{attribute 'reflection'} 
FUNCTION_BLOCK FB_WorkerDefGrid_Python EXTENDS FB_WorkerDefGrid IMPLEMENTS I_DeformationHandler
VAR_INPUT
END_VAR
VAR_OUTPUT
END_VAR
VAR
  // interface to py script
  fbPythonInterface : FB_PythonInterface;
  // references
  _iParamMediator : I_ParamMediator;
  
  // local copy of setttings
  _bNewJob : BOOL;  // new job was activated
  _CamGridSettings : ST_CameraGridSettings;
  _DefGridSettings : ST_DefGridSettings;
  
  // local copy of job setting
  _aJobName         : T_MaxString;
  _aJobGuid         : T_MaxString;
  _fImageWidthM     : LREAL;          // image width in [m]
  _fImageDepthM     : LREAL;          // image depth in [m]
  

  // messages
  fbMsg_PythonNotRunning : FB_MESSAGE;
END_VAR

VAR CONSTANT
  fC_DEFAULT_WOKER_POSITION : LREAL := 0.01;      // default worker position in [m]
END_VAR

METHOD PROTECTED  Attach : BOOL
VAR_INPUT
  iCT              : I_CT;                         (*container at triggered event position*)
END_VAR
VAR
  pCt : POINTER TO FB_ContainerDefGrid;
END_VAR
Attach := FALSE;
IF SUPER^.Attach(iCT:=iCT) THEN
  // OK, attached (enabled, was ok to be attached)
  IF getCtInst(iCT:=iCT, pCT=>pCt) = 0 THEN    // get specific container
    RETURN;
  END_IF
  
  // setup check
  IF _iParamMediator = 0 THEN Release(iCT:=iCT); LogError('Invalid param mediator'); RETURN; END_IF
  
  // Additional worker checks
  // - do we have a valid job? used mode?
  IF _CamGridSettings.eCameraMode > E_CameraMode.NoCorrection AND (iCT.pJob = 0 OR NOT _bJobActive) THEN
    pCt^.AbortDeformation(sReason:='No valid job', Src:=_pEcSrc^);
     Release(iCT:=iCT);
     
  ELSIF _CamGridSettings.eCameraMode > E_CameraMode.NoCorrection THEN
    // OK attach
    // -- only create ct if a deformation is active
    IF CreateDefCt(iCT:=iCT) THEN
        // set state
        pCt^.StartScript(iDeformationHandler:=THIS^);
        // attached
        Attach := TRUE;
    END_IF
  ELSE
    ; // ignore attach
  END_IF
ELSE
  // parent attach failed
END_IF
END_METHOD

(*
  Create/Release virtual ct in deformation handlers.
  :return: TRUE if success
*)
METHOD PRIVATE CreateDefCt : BOOL;
VAR_INPUT
  iCT : I_CT;
END_VAR
IF iCT = 0 THEN RETURN; END_IF

IF _CamGridSettings.eCameraMode >= E_CameraMode.Live THEN
  IF fbPythonInterface.RegisterCT(iCT.pCT^.nMemIndex) THEN
    CreateDefCt := TRUE;
  ELSE
    _pAttachedCt^.AbortDeformation(sReason:='Could not register to script', Src:=_pEcSrc^);
  END_IF
ELSE
  CreateDefCt := TRUE;
END_IF
END_METHOD

METHOD DeleteCachedCt : BOOL
VAR_INPUT
	iCT	: I_CT;
END_VAR
DeleteDefCt(iCT:=iCT);
END_METHOD

(*
  Delete/Release virtual ct in deformation handlers.
  :return: TRUE if sucess
*)
METHOD DeleteDefCt : BOOL
VAR_INPUT
  iCT : I_CT;
END_VAR
IF iCT = 0 THEN RETURN; END_IF

IF _CamGridSettings.eCameraMode >= E_CameraMode.Live THEN
  IF fbPythonInterface.RemoveCT(iCT.pCT^.nMemIndex) THEN
    DeleteDefCt := TRUE;
  ELSE
    LogError('Could not delete ct in script');
  END_IF
END_IF
END_METHOD

METHOD Init
VAR_INPUT
  iWorkerParams : I_WorkerParams;
  pMsgConfig : POINTER TO ST_MSG_CONFIG;         // message config
  fPrintResolution : LREAL := 1;                 // print(head) resolution in [dpi]
  fSubPxResolution : LREAL := 1;                 // SubPixel resolution [SubPx], resolution factor (fI_PrintResolution*fI_SubPxResolution=>Output resolution)
  bParallelCT : BOOL;                            // Support parallel processing of CTs
END_VAR
SUPER^.Init(iWorkerParams:=iWorkerParams, pMsgConfig:=pMsgConfig, fPrintResolution:=fPrintResolution, fSubPxResolution:=fSubPxResolution, bParallelCT:=bParallelCT);

// Init messages
fbMsg_PythonNotRunning.pI_MsgConfig := _pMsgConfigExt;
fbMsg_PythonNotRunning.iI_MsgLocation := ePr_BLK_PU;
fbMsg_PythonNotRunning.iI_MsgNumber := eC_DMAX_DEF_SCRIPT_NOT_RUNNING;
END_METHOD

METHOD InitWorkerPython
VAR_INPUT
  aScriptPath : T_MaxString;                     // path to cmd scripts
  //aAmsLocalHost : T_AmsNetID;                    // Ams netId localhost of the pc to run the script
  iDefGridParamMediator : I_ParamMediator;
END_VAR
IF NOT bInitialized OR _iWorkerParams.pCTManager = 0 THEN LogError('Base Worker not initialized! call init() before'); RETURN; END_IF
IF iDefGridParamMediator = 0 THEN bInitialized := FALSE; LogError('Invalid parameter, no valid param mediator'); RETURN; END_IF

// worker specific init
_iParamMediator := iDefGridParamMediator;

fbPythonInterface.Init(
  sCTManagerPath := _iWorkerParams.pCTManager^.sCTDefGridInstancesPath, 
  sScriptPath:=aScriptPath
);
END_METHOD

METHOD mJobStart
VAR_INPUT
	sJobDef	: CalmarCompPrint.I_JobDefinition;
END_VAR
// checks and fix defaults
IF _iParamMediator = 0 THEN LogError('JobStart: invalid parameter configuration'); RETURN; END_IF
IF _fWorkerPosition = 0 THEN _fWorkerPosition := fC_DEFAULT_WOKER_POSITION; LogError(F_Concat3(_name, ': worker position not set, set default=', TO_STRING(fC_DEFAULT_WOKER_POSITION))); END_IF

// configure
_aJobName := sJobDef.aJobName;
_aJobGuid := sJobDef.aJobId;
_fImageDepthM := sJobDef.fImageDepth/1000;
_fImageWidthM := sJobDef.fImageWidth/1000;

_bNewJob := TRUE;
_bJobActive := TRUE;
END_METHOD

METHOD  mJobStop
VAR_INPUT
	sStatus	: CalmarCompPrint.I_JobStatus;
END_VAR
fbPythonInterface.JobStop();
_bJobActive := FALSE;
END_METHOD

METHOD setupPosition
// !!! No Auto-Setup implemented 


(*
IF _pAttachedCt <> 0 THEN RETURN; END_IF    // Update only without attached container

fPosition := xyz + _fPmPosition;
*)
END_METHOD

METHOD  work
VAR_INPUT
END_VAR
VAR
  i : UDINT;
  tempCt  : POINTER TO FB_ContainerDefGrid;
  bDeformationDone : BOOL;
  bDeformationError : BOOL;
END_VAR
VAR_INST
  rT_EnablePyIf  : R_TRIG;
END_VAR
SUPER^.work();

IF _iParamMediator <> 0 THEN F_Report_Error(ErrType:=EN_REPORT_ERROR_TYPE.Report_Error_0Pointer); RETURN; END_IF
_CamGridSettings := _iParamMediator.sCameraGridSettings;
_DefGridSettings := _iParamMediator.sDeformationGridSetttings;

setupPosition();    // Worker position update

// reconfig script after job started (Mediator parameter are defined in JobStart())
IF _bNewJob OR rT_EnablePyIf.Q THEN   // new job activated or re-enabled
  _bNewJob := FALSE;
  
  // setup script
  fbPythonInterface.JobStart(
    aJobName:=_aJobName,
    aJobGuid:=_aJobGuid,
    nJobImageWidth:=DINT_TO_UDINT(F_MeterToSubPixel(fPosMeter:=_fImageDepthM, fResoSubPx:=_fPrintResolution)),
    nJobImageHeigth:=DINT_TO_UDINT(F_MeterToSubPixel(fPosMeter:=_fImageWidthM, fResoSubPx:=_fPrintResolution)),
    nCamFrameWidth:=DINT_TO_UDINT(FC_LREAL_TO_DINT(_CamGridSettings.fGridFeaturePitch)),
    pGridSettings:=ADR(_DefGridSettings)
  );
END_IF

// start/stop script
IF _CamGridSettings.eCameraMode >= E_CameraMode.Live AND THIS^.bWorkerEnable THEN 
  fbPythonInterface.bEnable := TRUE;
ELSE
  fbPythonInterface.bEnable := FALSE;
END_IF
rT_EnablePyIf(CLK:=fbPythonInterface.bEnable);

fbPythonInterface();

IF _pAttachedCt <> 0 THEN
  // nothing to do anymore just release CT
  // NOTE: the delete of the CT is done by DeleteDefCt() method directly into fbPythonInterface
  Release(_pAttachedCt^);
END_IF

// messages
fbMsg_PythonNotRunning(bI_Status:=fbPythonInterface.bError);
IF fbMsg_PythonNotRunning.bMsgAck THEN fbPythonInterface.ackError(); END_IF
END_METHOD

END_FUNCTION_BLOCK

(* stored: Version 1.1.0.1, ProductVersion 3.1.4024.11
   POU FB_WorkerDefGrid_Python: Id {da715aa5-d637-40ab-8d33-e404e3b6a6f1}, SpecialFunc None
   Folder I_DeformationHandler: Id {ceaf56cc-d085-4a2b-a063-c0fa29cdf9f9}
   Folder I_PrintStatusClient: Id {f883ee39-a8eb-4a93-9829-26e2a724ffe3}
   Method Attach: Id {42eaf325-ff4e-48df-be91-9b20bce3da44}
   Method CreateDefCt: Id {bdf419b5-1889-4837-99cf-ef4a36422f29}
   Method DeleteCachedCt: Id {0747863f-1393-4933-afe3-0c0b74eb26c2}
   Method DeleteDefCt: Id {1250acd3-857f-4045-a296-4dd4aaa257e9}
   Method Init: Id {f68f2ec1-c6b3-4670-a09a-c2c908e7b5dc}
   Method InitWorkerPython: Id {343b3a60-1392-4b26-a0f9-056258434c15}
   Method mJobStart: Id {0fd0f7ed-3d4d-47aa-ba8e-6404bd51c209}
   Method mJobStop: Id {db89a0b9-8d28-4bf7-9778-94d597d27cae}
   Method setupPosition: Id {306e6870-fcda-49b6-bbc8-487fc586e0b2}
   Method work: Id {3c4c9ab8-eeba-4bde-9db0-7737c05146ce} *)
